FUNCTION_BLOCK FB_SimpleTcpTaskQueue2
VAR_INPUT
END_VAR
VAR_OUTPUT
END_VAR
VAR
	ActingQueue			: FB_MemRingBufferEx;
	ArrActingQueue		: ARRAY[0..MAXBUFFERSIZE] OF ST_TcpTaskBuffer2;
	
	fbMemMan			: FB_DynMem_Manager2;
	
	PushTask	: ST_TcpTask2;
	PullTask	: ST_TcpTask2;
	EmptyTask	: ST_TcpTask2;
	
	StepTaskConsume : DINT;
	
	_NoTaskToConsume : BOOL;
	_WaitingForTaskDone: BOOL;
	_ActingTaskCount: UDINT;
	_ActingUsedSize: UDINT;
	_ActingFreeSize: UDINT;
END_VAR
VAR CONSTANT
	MAXBUFFERSIZE: UDINT := 128;
END_VAR

_CyclicLogic();

METHOD PROTECTED _CyclicLogic : BOOL
VAR_INPUT
END_VAR
(* 获取队列负载数据 *)
ActingQueue.A_GetFreeSize(pWrite:= , cbWrite:= , pBuffer:= ADR(ArrActingQueue), cbBuffer:= SIZEOF(ArrActingQueue), 
	bOk=> , pRead=> , cbRead=> , nCount=> _ActingTaskCount, cbSize=> _ActingUsedSize, cbFree=> _ActingFreeSize);
(* 状态显示 *)
_NoTaskToConsume := (StepTaskConsume = 0);
_WaitingForTaskDone := (StepTaskConsume <> 0);
(* 如果队列中有事件，取出事件并等待Finish *)
CASE StepTaskConsume OF
	0:
	_NoTaskToConsume := TRUE;
	IF ActingQueue.nCount <> 0 THEN
		StepTaskConsume := 10;
	END_IF
	
	10:
	ActingQueue.A_GetHead(pWrite:= , cbWrite:= , pBuffer:= ADR(ArrActingQueue), cbBuffer:= SIZEOF(ArrActingQueue), 
	bOk=> , pRead=> , cbRead=> , nCount=> _ActingTaskCount, cbSize=> _ActingUsedSize, cbFree=> _ActingFreeSize);
	IF ActingQueue.bOk THEN
		MEMCPY(destAddr:= ADR(PullTask), srcAddr:= ActingQueue.pRead, n:= MIN(SIZEOF(PullTask),ActingQueue.cbRead));
		StepTaskConsume := 20;
	ELSE
		StepTaskConsume := 0;
		ADSLOGSTR(msgCtrlMask:= ADSLOG_MSGTYPE_ERROR OR ADSLOG_MSGTYPE_STRING,
			msgFmtStr:= 'CyclicLogic: FIFO gethead failed', strArg:= '');
	END_IF
	
	20:
	// wait for task done
	
END_CASE
END_METHOD

PROPERTY ActingFreeSize : UDINT
GET
ActingFreeSize := _ActingFreeSize;
END_GET
END_PROPERTY

PROPERTY ActingTaskCount : UDINT
GET
ActingTaskCount := _ActingTaskCount;
END_GET
END_PROPERTY

PROPERTY ActingUsedSize : UDINT
GET
ActingUsedSize := _ActingUsedSize;
END_GET
END_PROPERTY

METHOD AddActingTask : BOOL
VAR_INPUT
	TaskName : STRING(24);
	TaskType : INT; (* 0:Once, 1:Regular *)
	pData : PVOID;
	nData : UDINT;
END_VAR
VAR
	pDynMem : PVOID;
END_VAR
IF nData > ActingQueue.cbFree THEN
	ADSLOGSTR(msgCtrlMask:= ADSLOG_MSGTYPE_ERROR OR ADSLOG_MSGTYPE_STRING,
		msgFmtStr:= 'AddTaskFailed: No free space in FIFO', strArg:= '');
	RETURN;
END_IF
pDynMem := fbMemMan.Alloc(nSize:= nData, bReset:= TRUE);
IF pDynMem = 0 THEN
	ADSLOGSTR(msgCtrlMask:= ADSLOG_MSGTYPE_ERROR OR ADSLOG_MSGTYPE_STRING,
		msgFmtStr:= 'AddTaskFailed: Allocate memory failed', strArg:= '');
	RETURN;
END_IF
MEMCPY(destAddr:= pDynMem, srcAddr:= pData, n:= nData);
PushTask.TaskName := TaskName;
PushTask.TaskType := TaskType;
PushTask.pData := pDynMem;
PushTask.nData := nData;
ActingQueue.A_AddTail(pWrite:= ADR(PushTask), cbWrite:= SIZEOF(PushTask), pBuffer:= ADR(ArrActingQueue), cbBuffer:= SIZEOF(ArrActingQueue), 
	bOk=> AddActingTask, pRead=> , cbRead=> , nCount=> _ActingTaskCount, cbSize=> _ActingUsedSize, cbFree=> _ActingFreeSize);
IF ActingQueue.bOk THEN
	AddActingTask := TRUE;
ELSE
	ADSLOGSTR(msgCtrlMask:= ADSLOG_MSGTYPE_ERROR OR ADSLOG_MSGTYPE_STRING,
		msgFmtStr:= 'AddTaskFailed: FIFO addtail failed ', strArg:= '');
	fbMemMan.Free2(pDynMem);
END_IF
END_METHOD

PROPERTY CurrentTask : ST_TcpTask2
GET
CurrentTask := PullTask;
END_GET
END_PROPERTY

METHOD FinishTask : BOOL
VAR_INPUT
END_VAR
VAR
	pDynMem : PVOID;
END_VAR
(* 调用freehead，释放FIFO头，判断释放是否成功 *)
ActingQueue.A_FreeHead(pWrite:= , cbWrite:= , pBuffer:= ADR(ArrActingQueue), cbBuffer:= SIZEOF(ArrActingQueue), 
	bOk=> , pRead=> , cbRead=> , nCount=> _ActingTaskCount, cbSize=> _ActingUsedSize, cbFree=> _ActingFreeSize);
IF ActingQueue.bOk THEN
	IF ActingQueue.nCount <> 0 THEN
		StepTaskConsume := 10;
	ELSE
		StepTaskConsume := 0;
	END_IF
ELSE
	ADSLOGSTR(msgCtrlMask:= ADSLOG_MSGTYPE_ERROR OR ADSLOG_MSGTYPE_STRING,
		msgFmtStr:= 'FinishTaskFailed: FIFO freehead failed', strArg:= '');
	RETURN;
END_IF

FinishTask := TRUE;
pDynMem := PullTask.pData;
PullTask := EmptyTask;
//MEMCPY(destAddr:= ADR(PullTask), srcAddr:= ADR(EmptyTask), n:= SIZEOF(PullTask));
fbMemMan.Free2(pDynMem);
END_METHOD

PROPERTY NoTaskToConsume : BOOL
GET
NoTaskToConsume := _NoTaskToConsume;
END_GET
END_PROPERTY

PROPERTY WaitingForTaskDone : BOOL
GET
WaitingForTaskDone := _WaitingForTaskDone;
END_GET
END_PROPERTY

END_FUNCTION_BLOCK

(* stored: Version 1.1.0.1, ProductVersion 3.1.4024.12
   POU FB_SimpleTcpTaskQueue2: Id {38af2dbd-f972-4e1b-92b0-127bd0bd71aa}, SpecialFunc None
   Method _CyclicLogic: Id {a28a799e-f312-4bf4-9a26-4d2912a197eb}
   Property ActingFreeSize: Id {4a11dcf3-37ae-47a6-a60d-15ca4d3d6b5c}
   Get Get: Id {e79b8cb3-4f79-4ab0-8579-14055ee0e5ac}
   Property ActingTaskCount: Id {c9bce407-85f3-49a4-ad74-915784102de5}
   Get Get: Id {0ba26ec7-46e2-4029-b304-8274a94a93f9}
   Property ActingUsedSize: Id {5368d4b7-3fb1-45b2-b2df-9a628280ac7c}
   Get Get: Id {d7cf890d-a5fb-48e8-af7b-222abf70736d}
   Method AddActingTask: Id {be0719ae-69cb-4aa2-aab1-f53d0c2a7e85}
   Property CurrentTask: Id {c15abde0-ae8c-4d5c-b639-9399f4b83c10}
   Get Get: Id {6d395937-af01-41e8-bb47-334095f8a881}
   Method FinishTask: Id {04bb83a5-74c0-4aa1-b8db-ac16a729fb64}
   Property NoTaskToConsume: Id {2bd7de61-47c8-4fe9-a18d-79c11b9ccb37}
   Get Get: Id {aa3b4586-d911-457b-a696-0ff22495f475}
   Property WaitingForTaskDone: Id {275fb84f-a593-4e1a-a76b-f86ad83c524f}
   Get Get: Id {ee981d17-1211-43cb-b757-ebf937181454} *)
